(* PLC project Unnamed, Unknown Unnamed 1 *)
(* stored: creationDateTime 2019-08-06T14:23:42, modificationDateTime 2024-03-26T14:11:47 *)

PROGRAM MainStuff
  VAR
    LocalVar0 : DINT;
    LocalVar1 : DINT;
  END_VAR

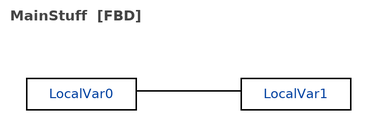
(* FBD diagram, written out as Structured Text *)
LocalVar1 := LocalVar0;
END_PROGRAM

CONFIGURATION config
  RESOURCE resource1 ON PLC
    TASK task0(INTERVAL := T#20ms, PRIORITY := 0);
    PROGRAM instance0 WITH task0 : MainStuff;
  END_RESOURCE
END_CONFIGURATION
